FUNCTION_BLOCK ME_ThreeConCtl (* Composite Function Block Type *)
  (* Standard: 61499-2 *)
  (* Version 0.2, 2003-12-05, JHC, Rockwell Automation, Renamed from NEWCOMPFB. *)
  (* Version 0.1, 2002-01-08, JHC, Rockwell Automation, Added DLY FB as example. *)
  (* Version 0.0, 2000-05-27, JHC, Rockwell Automation *)
  (* Compiler header: package fb.rt.cs725; *)
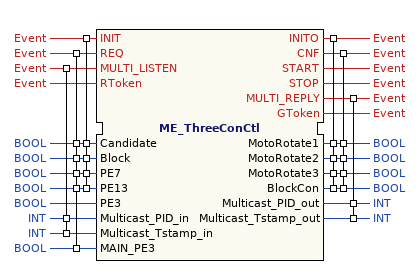
  EVENT_INPUT
    INIT WITH Candidate, Block, PE7, PE13; (* Initialization Request *)
    REQ WITH Block, Candidate, PE7, MAIN_PE3, PE13; (* Normal Execution Request *)
    MULTI_LISTEN WITH Multicast_PID_in, Multicast_Tstamp_in;
    RToken;
  END_EVENT
  EVENT_OUTPUT
    INITO WITH MotoRotate1, MotoRotate2, MotoRotate3, BlockCon; (* Initialization Confirm *)
    CNF WITH MotoRotate1, MotoRotate2, MotoRotate3, BlockCon; (* Execution Confirmation *)
    START;
    STOP;
    MULTI_REPLY WITH Multicast_PID_out, Multicast_Tstamp_out;
    GToken;
  END_EVENT
  VAR_INPUT
    Candidate : BOOL;
    Block : BOOL;
    PE7 : BOOL;
    PE13 : BOOL;
    PE3 : BOOL;
    Multicast_PID_in : INT;
    Multicast_Tstamp_in : INT;
    MAIN_PE3 : BOOL;
  END_VAR
  VAR_OUTPUT
    MotoRotate1 : BOOL;
    MotoRotate2 : BOOL;
    MotoRotate3 : BOOL;
    BlockCon : BOOL;
    Multicast_PID_out : INT;
    Multicast_Tstamp_out : INT;
  END_VAR
  FBS
    FC11 : Conveyor_7;
    FC13 : ConveyorCTL(PE := 0, Block := 0, Candidate := 0);
    Multicast_FC12_Three : MulticastConveyorCTL(Candidate := 0, Block := 0, MyPID := 20, MyTstamp := 0, MyLoadDelay := 5);
  END_FBS
  EVENT_CONNECTIONS
    INIT TO FC11.INIT;
    REQ TO FC11.REQ;
    FC13.INITO TO INITO;
    FC13.CNF TO CNF;
    FC11.STOP TO STOP;
    FC11.START TO START;
    REQ TO FC13.REQ;
    FC11.CNF TO CNF;
    MULTI_LISTEN TO Multicast_FC12_Three.LISTEN;
    Multicast_FC12_Three.REPLY TO MULTI_REPLY;
    REQ TO Multicast_FC12_Three.REQ;
    Multicast_FC12_Three.CNF TO CNF;
    FC11.INITO TO Multicast_FC12_Three.INIT;
    Multicast_FC12_Three.INITO TO FC13.INIT;
    RToken TO FC11.RToken;
    FC11.GToken TO GToken;
    FC13.STOP TO Multicast_FC12_Three.CAS_STOP;
    FC13.START TO Multicast_FC12_Three.CAS_START;
    Multicast_FC12_Three.STOP TO FC11.CAS_STOP;
    Multicast_FC12_Three.START TO FC11.CAS_START;
  END_CONNECTIONS
  DATA_CONNECTIONS
    FC13.MotoRotate TO MotoRotate3;
    FC11.MotoRotate TO MotoRotate1;
    PE7 TO FC11.PE;
    Block TO FC11.Block;
    FC11.BlockCon TO BlockCon;
    Candidate TO FC11.Candidate;
    Multicast_FC12_Three.MotoRotate TO MotoRotate2;
    Multicast_PID_in TO Multicast_FC12_Three.PID_in;
    Multicast_Tstamp_in TO Multicast_FC12_Three.Tstamp_in;
    Multicast_FC12_Three.Tstamp_out TO Multicast_Tstamp_out;
    Multicast_FC12_Three.PID_out TO Multicast_PID_out;
    PE3 TO Multicast_FC12_Three.PE;
    MAIN_PE3 TO Multicast_FC12_Three.MAIN_PE;
    PE13 TO FC11.PE_13;
  END_CONNECTIONS
END_FUNCTION_BLOCK
